ABB RAPID module: Wobj_wobj_B1.mod

MODULE Wobj_wobj_B1
	! Points are read in order of declaration.
  ! Please do not change the order of points!

  LOCAL PERS robtarget pWobj_U_PointX1:=[[-42.42045,-2235.461,-607.6553],[0.00631720200181007,-0.720873773097992,0.69301700592041,-0.00533610209822655],[-2,0,1,0],[0,9E+09,9E+09,9E+09,9E+09,9E+09]];
	LOCAL PERS robtarget pWobj_U_PointX2:=[[448.1077,-2215.543,-605.6558],[0.00631724949926138,-0.720873773097992,0.69301700592041,-0.00533630838617682],[-1,0,2,0],[0,9E+09,9E+09,9E+09,9E+09,9E+09]];
	LOCAL PERS robtarget pWobj_U_PointY1:=[[-59.42518,-1697.987,-605.6547],[0.00631762156262994,-0.720876038074493,0.693014681339264,-0.00533577846363187],[-2,0,1,0],[0,9E+09,9E+09,9E+09,9E+09,9E+09]];

ENDMODULE
